// Mitsubishi GX Works2 project: Melsec   PLC: FX3U/FX3UC

PROGRAM MAIN
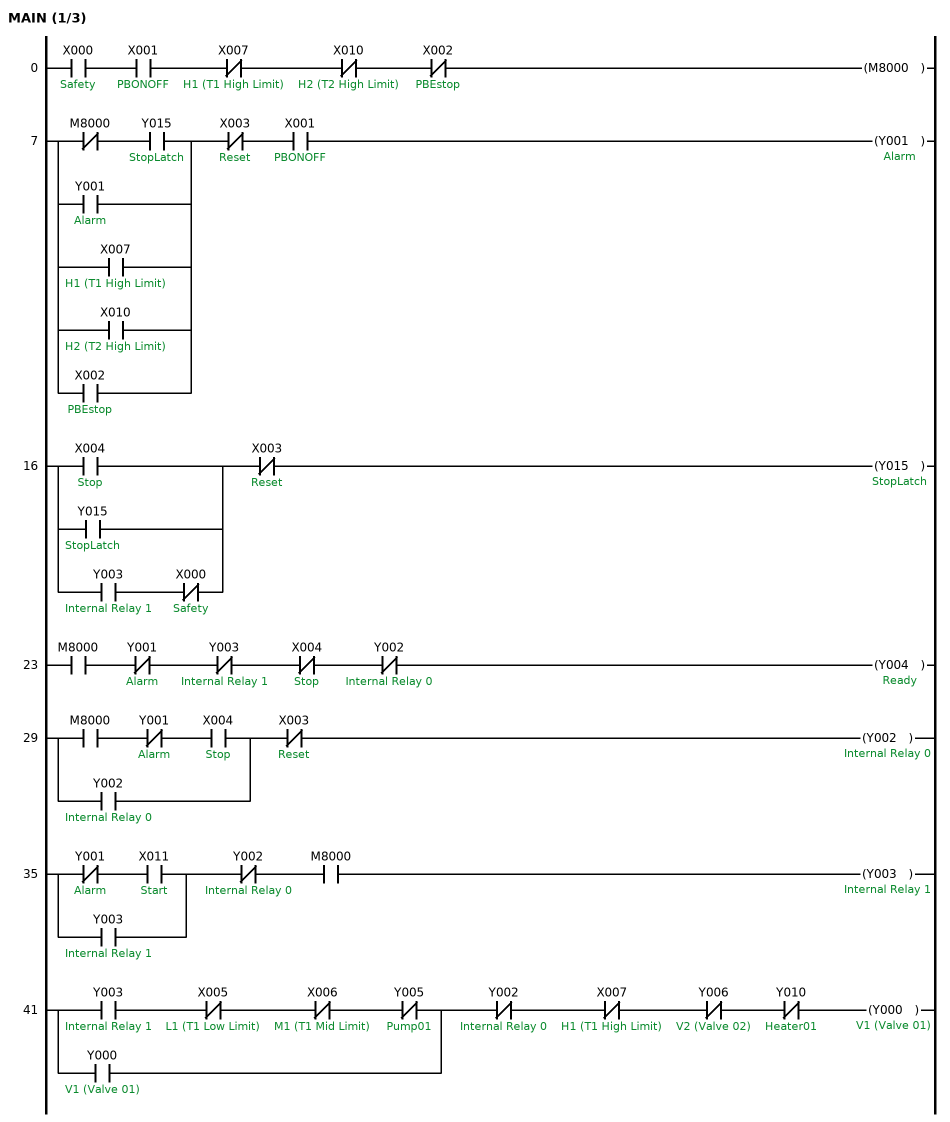
0     LD      X000  ; Safety
      AND     X001  ; PBONOFF
      ANI     X007  ; H1 (T1 High Limit)
      ANI     X010  ; H2 (T2 High Limit)
      ANI     X002  ; PBEstop
      OUT     M8000
7     LDI     M8000
      AND     Y015  ; StopLatch
      OR      Y001  ; Alarm
      OR      X007  ; H1 (T1 High Limit)
      OR      X010  ; H2 (T2 High Limit)
      OR      X002  ; PBEstop
      ANI     X003  ; Reset
      AND     X001  ; PBONOFF
      OUT     Y001  ; Alarm
16    LD      X004  ; Stop
      OR      Y015  ; StopLatch
      LD      Y003  ; Internal Relay 1
      ANI     X000  ; Safety
      ORB
      ANI     X003  ; Reset
      OUT     Y015  ; StopLatch
23    LD      M8000
      ANI     Y001  ; Alarm
      ANI     Y003  ; Internal Relay 1
      ANI     X004  ; Stop
      ANI     Y002  ; Internal Relay 0
      OUT     Y004  ; Ready
29    LD      M8000
      ANI     Y001  ; Alarm
      AND     X004  ; Stop
      OR      Y002  ; Internal Relay 0
      ANI     X003  ; Reset
      OUT     Y002  ; Internal Relay 0
35    LDI     Y001  ; Alarm
      AND     X011  ; Start
      OR      Y003  ; Internal Relay 1
      ANI     Y002  ; Internal Relay 0
      AND     M8000
      OUT     Y003  ; Internal Relay 1
41    LD      Y003  ; Internal Relay 1
      ANI     X005  ; L1 (T1 Low Limit)
      ANI     X006  ; M1 (T1 Mid Limit)
      ANI     Y005  ; Pump01
      OR      Y000  ; V1 (Valve 01)
      ANI     Y002  ; Internal Relay 0
      ANI     X007  ; H1 (T1 High Limit)
      ANI     Y006  ; V2 (Valve 02)
      ANI     Y010  ; Heater01
      OUT     Y000  ; V1 (Valve 01)
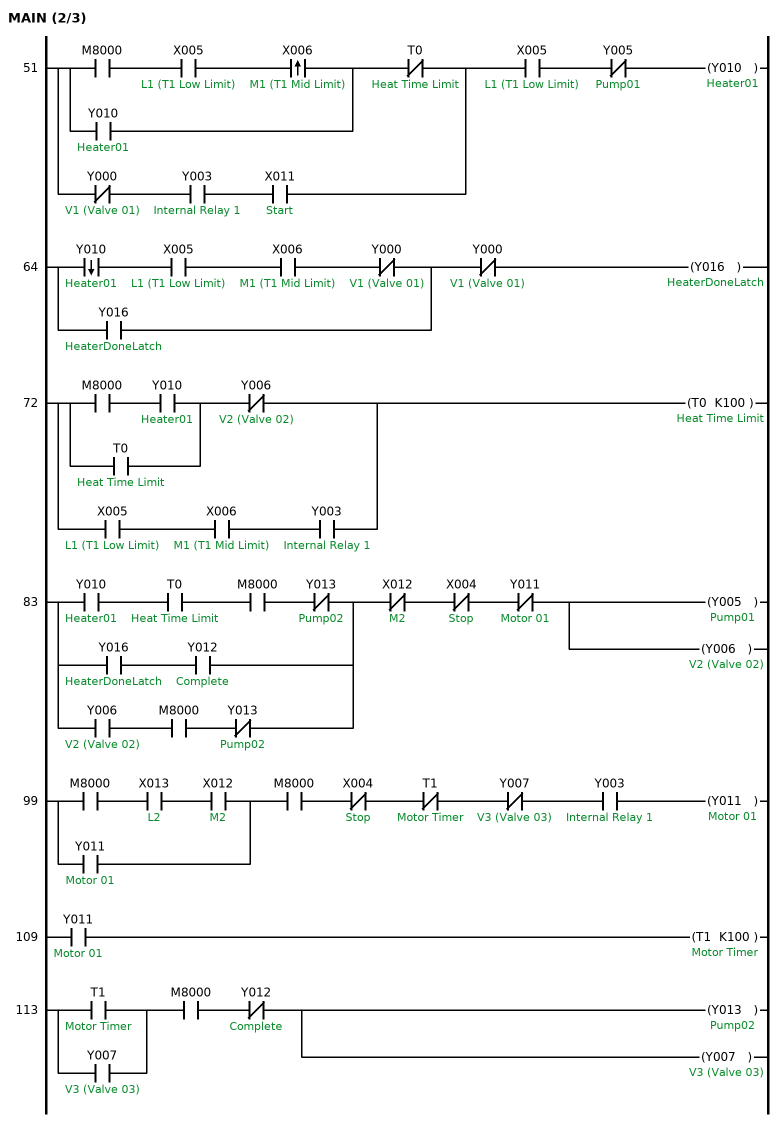
51    LD      M8000
      AND     X005  ; L1 (T1 Low Limit)
      ANDP    X006  ; M1 (T1 Mid Limit)
      OR      Y010  ; Heater01
      ANI     T0  ; Heat Time Limit
      LDI     Y000  ; V1 (Valve 01)
      AND     Y003  ; Internal Relay 1
      AND     X011  ; Start
      ORB
      AND     X005  ; L1 (T1 Low Limit)
      ANI     Y005  ; Pump01
      OUT     Y010  ; Heater01
64    LDF     Y010  ; Heater01
      AND     X005  ; L1 (T1 Low Limit)
      AND     X006  ; M1 (T1 Mid Limit)
      ANI     Y000  ; V1 (Valve 01)
      OR      Y016  ; HeaterDoneLatch
      ANI     Y000  ; V1 (Valve 01)
      OUT     Y016  ; HeaterDoneLatch
72    LD      M8000
      AND     Y010  ; Heater01
      OR      T0  ; Heat Time Limit
      ANI     Y006  ; V2 (Valve 02)
      LD      X005  ; L1 (T1 Low Limit)
      AND     X006  ; M1 (T1 Mid Limit)
      AND     Y003  ; Internal Relay 1
      ORB
      OUT     T0 K100  ; Heat Time Limit
83    LD      Y010  ; Heater01
      AND     T0  ; Heat Time Limit
      AND     M8000
      ANI     Y013  ; Pump02
      LD      Y016  ; HeaterDoneLatch
      AND     Y012  ; Complete
      ORB
      LD      Y006  ; V2 (Valve 02)
      AND     M8000
      ANI     Y013  ; Pump02
      ORB
      ANI     X012  ; M2
      ANI     X004  ; Stop
      ANI     Y011  ; Motor 01
      OUT     Y005  ; Pump01
      OUT     Y006  ; V2 (Valve 02)
99    LD      M8000
      AND     X013  ; L2
      AND     X012  ; M2
      OR      Y011  ; Motor 01
      AND     M8000
      ANI     X004  ; Stop
      ANI     T1  ; Motor Timer
      ANI     Y007  ; V3 (Valve 03)
      AND     Y003  ; Internal Relay 1
      OUT     Y011  ; Motor 01
109   LD      Y011  ; Motor 01
      OUT     T1 K100  ; Motor Timer
113   LD      T1  ; Motor Timer
      OR      Y007  ; V3 (Valve 03)
      AND     M8000
      ANI     Y012  ; Complete
      OUT     Y013  ; Pump02
      OUT     Y007  ; V3 (Valve 03)
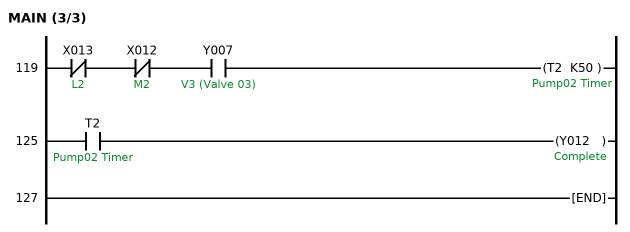
119   LDI     X013  ; L2
      ANI     X012  ; M2
      AND     Y007  ; V3 (Valve 03)
      OUT     T2 K50  ; Pump02 Timer
125   LD      T2  ; Pump02 Timer
      OUT     Y012  ; Complete
127   END
END_PROGRAM

// device comments not shown above
Y014  ; HeatLatch
M4000  ; Internal Safety Relay
